(*
SPDX-FileCopyrightText: © 2026 Oleksandr Tiutyk <trofimich@gmail.com>
SPDX-License-Identifier: MIT
License: https://opensource.org/license/mit
*)

(*!
<summary>Provides this library's namespace text to object metadata getters.</summary>
<description>
Owns the namespace extractor for the program instance's lifetime; no cyclic execution is required.
</description>
*)

{attribute 'no_explicit_call' := 'do not call this POU directly'}
PROGRAM INTERNAL CurrentNamespace
VAR
	{attribute 'hide'} 
	_NamespaceExtractor : NamespaceExtractor;
END_VAR

{attribute 'monitoring' := 'call'}
(*!
<summary>Returns a borrowed reference to the stored namespace text.</summary>
<description>
The reference belongs to this program instance and remains valid while it exists. Callers must treat the text
as read-only; reading does not copy or allocate storage.
</description>
*)
PROPERTY Name : REFERENCE TO STRING
GET
Name REF= _NamespaceExtractor.CurrentNamespace;
END_GET
END_PROPERTY

END_PROGRAM

(* stored: Version 1.1.0.1
   POU CurrentNamespace: Id {6352a046-3db4-4588-9020-8c47a4e3d2b0}, SpecialFunc None
   Property Name: Id {e73030d0-3401-44c9-8168-4bca8004bdd1}
   Get Get: Id {375ab72f-5a5f-4acb-8873-b22a2cd7a60c} *)
